{attribute 'qualified_only'}
{attribute 'strict'}
TYPE AutostoreControlCommand :
(
	DO_NOTHING := 0,
	START	:= 1,
	STOP	:= 2
);
END_TYPE

(* stored: Version 1.1.0.1, ProductVersion 3.1.4024.12
   DUT AutostoreControlCommand: Id {92c937d9-f38e-456a-a4fc-df36484f4ae0} *)
